PROGRAM PRG_1_PlcTask
VAR

END_VAR

PRG_MR1K1_BEND();
PRG_MR1K1_BEND_BENDER();
//PRG_MR1K2_SWITCH();
PRG_SP1K1_MONO();
//PRG_SL1K2_EXIT();
PRG_ST1K1_ZOS();
//PRG_DAQ_ENCODER();
//PRG_SPO_PMPS();
PRG_2_PMPS_POST();

PRG_ZeroOrder_PMPS();

END_PROGRAM

(* stored: Version 1.1.0.1, ProductVersion 3.1.4022.12
   POU PRG_1_PlcTask: Id {21f3a158-4837-47ff-8ec7-29454a44967d}, SpecialFunc None *)
